// TIA Portal V20 export
// export: Created 2026-07-19T01:14:26.1398018Z, ExportSetting WithDefaults, DisplayName Totally Integrated Automation Portal, DisplayVersion V20 Update 5, DisplayName TIA Portal Openness, DisplayVersion V20 Update 4, DisplayName TIA Portal Version Control Interface, DisplayVersion V20 Update 5, DisplayName SINAMICS Startdrive Advanced, DisplayVersion V20, DisplayName SINAMICS DCC, DisplayVersion V20, DisplayName SINAMICS Startdrive G130, G150, S120, S150, SINAMICS MV, G220, S200, S210, DisplayVersion V20, DisplayName SINAMICS Startdrive G110M, G120, G120C, G120D, G120P, G115D, DisplayVersion V20, DisplayName STEP 7 Professional, DisplayVersion V20 Update 5, DisplayName STEP 7 Safety, DisplayVersion V20 Update 2, DisplayName WinCC Basic/Comfort/Advanced, DisplayVersion V20 Update 5, DisplayName WinCC Unified, DisplayVersion V20 Update 5
FUNCTION "HandAuthorSplitsMerges" : Void   // FC3, LAD
{ S7_Optimized_Access := 'TRUE' }
VERSION : 0.1
// stored: AutoNumber true, IsIECCheckEnabled false, SetENOAutomatically false, UDAEnableTagReadback false
   VAR_OUTPUT
      OutputVars : Array[0..10] of Bool;
   END_VAR
   VAR_TEMP   // added for the SCL form of the ladder/FBD networks
      _w1 : Bool;
      _w2 : Bool;
   END_VAR
BEGIN

REGION Network 1: Split Cascade
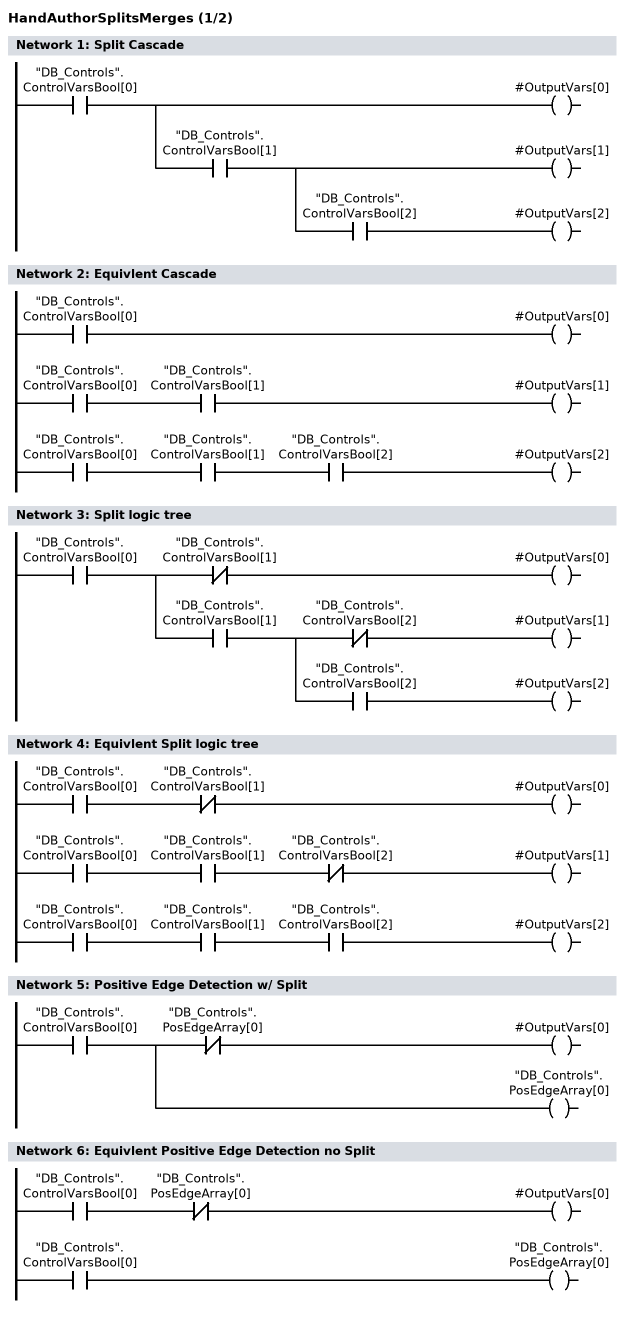
   RUNG wire#powerrail
      Contact( "DB_Controls".ControlVarsBool[0] )
      wire#w1
      Coil( #OutputVars[0] )
   END_RUNG
   RUNG wire#w1
      Contact( "DB_Controls".ControlVarsBool[1] )
      wire#w2
      Coil( #OutputVars[1] )
   END_RUNG
   RUNG wire#w2
      Contact( "DB_Controls".ControlVarsBool[2] )
      Coil( #OutputVars[2] )
   END_RUNG
   // the same network as SCL:
   #OutputVars[0] := "DB_Controls".ControlVarsBool[0];
   #OutputVars[1] := "DB_Controls".ControlVarsBool[0] AND "DB_Controls".ControlVarsBool[1];
   #OutputVars[2] := "DB_Controls".ControlVarsBool[0] AND "DB_Controls".ControlVarsBool[1] AND "DB_Controls".ControlVarsBool[2];
END_REGION

REGION Network 2: Equivlent Cascade
   RUNG wire#powerrail
      Contact( "DB_Controls".ControlVarsBool[0] )
      Coil( #OutputVars[0] )
   END_RUNG
   RUNG wire#powerrail
      Contact( "DB_Controls".ControlVarsBool[0] )
      Contact( "DB_Controls".ControlVarsBool[1] )
      Coil( #OutputVars[1] )
   END_RUNG
   RUNG wire#powerrail
      Contact( "DB_Controls".ControlVarsBool[0] )
      Contact( "DB_Controls".ControlVarsBool[1] )
      Contact( "DB_Controls".ControlVarsBool[2] )
      Coil( #OutputVars[2] )
   END_RUNG
   // the same network as SCL:
   #OutputVars[0] := "DB_Controls".ControlVarsBool[0];
   #OutputVars[1] := "DB_Controls".ControlVarsBool[0] AND "DB_Controls".ControlVarsBool[1];
   #OutputVars[2] := "DB_Controls".ControlVarsBool[0] AND "DB_Controls".ControlVarsBool[1] AND "DB_Controls".ControlVarsBool[2];
END_REGION

REGION Network 3: Split logic tree
   RUNG wire#powerrail
      Contact( "DB_Controls".ControlVarsBool[0] )
      wire#w1
      I_Contact( "DB_Controls".ControlVarsBool[1] )
      Coil( #OutputVars[0] )
   END_RUNG
   RUNG wire#w1
      Contact( "DB_Controls".ControlVarsBool[1] )
      wire#w2
      I_Contact( "DB_Controls".ControlVarsBool[2] )
      Coil( #OutputVars[1] )
   END_RUNG
   RUNG wire#w2
      Contact( "DB_Controls".ControlVarsBool[2] )
      Coil( #OutputVars[2] )
   END_RUNG
   // the same network as SCL:
   #OutputVars[0] := "DB_Controls".ControlVarsBool[0] AND NOT "DB_Controls".ControlVarsBool[1];
   #_w1 := "DB_Controls".ControlVarsBool[0] AND "DB_Controls".ControlVarsBool[1];
   #OutputVars[1] := #_w1 AND NOT "DB_Controls".ControlVarsBool[2];
   #OutputVars[2] := #_w1 AND "DB_Controls".ControlVarsBool[2];
END_REGION

REGION Network 4: Equivlent Split logic tree
   RUNG wire#powerrail
      Contact( "DB_Controls".ControlVarsBool[0] )
      I_Contact( "DB_Controls".ControlVarsBool[1] )
      Coil( #OutputVars[0] )
   END_RUNG
   RUNG wire#powerrail
      Contact( "DB_Controls".ControlVarsBool[0] )
      Contact( "DB_Controls".ControlVarsBool[1] )
      I_Contact( "DB_Controls".ControlVarsBool[2] )
      Coil( #OutputVars[1] )
   END_RUNG
   RUNG wire#powerrail
      Contact( "DB_Controls".ControlVarsBool[0] )
      Contact( "DB_Controls".ControlVarsBool[1] )
      Contact( "DB_Controls".ControlVarsBool[2] )
      Coil( #OutputVars[2] )
   END_RUNG
   // the same network as SCL:
   #OutputVars[0] := "DB_Controls".ControlVarsBool[0] AND NOT "DB_Controls".ControlVarsBool[1];
   #OutputVars[1] := "DB_Controls".ControlVarsBool[0] AND "DB_Controls".ControlVarsBool[1] AND NOT "DB_Controls".ControlVarsBool[2];
   #OutputVars[2] := "DB_Controls".ControlVarsBool[0] AND "DB_Controls".ControlVarsBool[1] AND "DB_Controls".ControlVarsBool[2];
END_REGION

REGION Network 5: Positive Edge Detection w/ Split
   RUNG wire#powerrail
      Contact( "DB_Controls".ControlVarsBool[0] )
      wire#w1
      I_Contact( "DB_Controls".PosEdgeArray[0] )
      Coil( #OutputVars[0] )
   END_RUNG
   RUNG wire#w1
      Coil( "DB_Controls".PosEdgeArray[0] )
   END_RUNG
   // the same network as SCL:
   #OutputVars[0] := "DB_Controls".ControlVarsBool[0] AND NOT "DB_Controls".PosEdgeArray[0];
   "DB_Controls".PosEdgeArray[0] := "DB_Controls".ControlVarsBool[0];
END_REGION

REGION Network 6: Equivlent Positive Edge Detection no Split
   RUNG wire#powerrail
      Contact( "DB_Controls".ControlVarsBool[0] )
      I_Contact( "DB_Controls".PosEdgeArray[0] )
      Coil( #OutputVars[0] )
   END_RUNG
   RUNG wire#powerrail
      Contact( "DB_Controls".ControlVarsBool[0] )
      Coil( "DB_Controls".PosEdgeArray[0] )
   END_RUNG
   // the same network as SCL:
   #OutputVars[0] := "DB_Controls".ControlVarsBool[0] AND NOT "DB_Controls".PosEdgeArray[0];
   "DB_Controls".PosEdgeArray[0] := "DB_Controls".ControlVarsBool[0];
END_REGION

REGION Network 7: Negitive Edge Detection /w split and merge
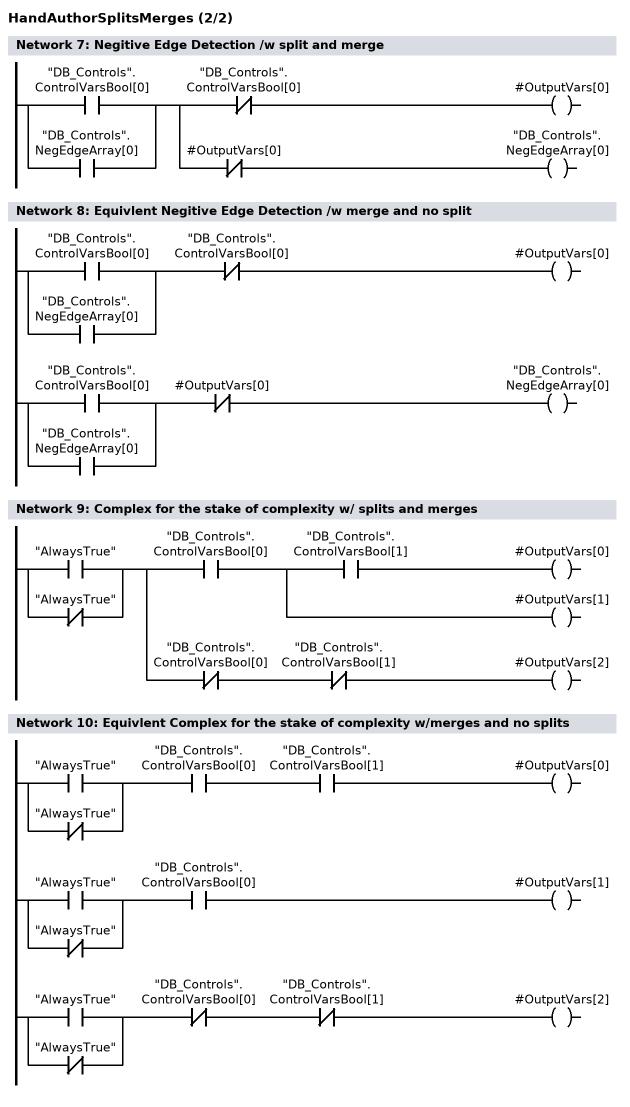
   RUNG wire#powerrail
      Contact( "DB_Controls".ControlVarsBool[0] )
      wire#w1
      I_Contact( "DB_Controls".ControlVarsBool[0] )
      Coil( #OutputVars[0] )
   END_RUNG
   RUNG wire#powerrail
      Contact( "DB_Controls".NegEdgeArray[0] )
   END_RUNG wire#w1
   RUNG wire#w1
      I_Contact( #OutputVars[0] )
      Coil( "DB_Controls".NegEdgeArray[0] )
   END_RUNG
   // the same network as SCL:
   #_w1 := "DB_Controls".ControlVarsBool[0] OR "DB_Controls".NegEdgeArray[0];
   #OutputVars[0] := #_w1 AND NOT "DB_Controls".ControlVarsBool[0];
   "DB_Controls".NegEdgeArray[0] := #_w1 AND NOT #OutputVars[0];
END_REGION

REGION Network 8: Equivlent Negitive Edge Detection /w merge and no split
   RUNG wire#powerrail
      Contact( "DB_Controls".ControlVarsBool[0] )
      wire#w1
      I_Contact( "DB_Controls".ControlVarsBool[0] )
      Coil( #OutputVars[0] )
   END_RUNG
   RUNG wire#powerrail
      Contact( "DB_Controls".NegEdgeArray[0] )
   END_RUNG wire#w1
   RUNG wire#powerrail
      Contact( "DB_Controls".ControlVarsBool[0] )
      wire#w2
      I_Contact( #OutputVars[0] )
      Coil( "DB_Controls".NegEdgeArray[0] )
   END_RUNG
   RUNG wire#powerrail
      Contact( "DB_Controls".NegEdgeArray[0] )
   END_RUNG wire#w2
   // the same network as SCL:
   #OutputVars[0] := ("DB_Controls".ControlVarsBool[0] OR "DB_Controls".NegEdgeArray[0]) AND NOT "DB_Controls".ControlVarsBool[0];
   "DB_Controls".NegEdgeArray[0] := ("DB_Controls".ControlVarsBool[0] OR "DB_Controls".NegEdgeArray[0]) AND NOT #OutputVars[0];
END_REGION

REGION Network 9: Complex for the stake of complexity w/ splits and merges
   RUNG wire#powerrail
      Contact( "AlwaysTrue" )
      wire#w1
      Contact( "DB_Controls".ControlVarsBool[0] )
      wire#w2
      Contact( "DB_Controls".ControlVarsBool[1] )
      Coil( #OutputVars[0] )
   END_RUNG
   RUNG wire#powerrail
      I_Contact( "AlwaysTrue" )
   END_RUNG wire#w1
   RUNG wire#w2
      Coil( #OutputVars[1] )
   END_RUNG
   RUNG wire#w1
      I_Contact( "DB_Controls".ControlVarsBool[0] )
      I_Contact( "DB_Controls".ControlVarsBool[1] )
      Coil( #OutputVars[2] )
   END_RUNG
   // the same network as SCL:
   #_w1 := "AlwaysTrue" OR NOT "AlwaysTrue";
   #_w2 := #_w1 AND "DB_Controls".ControlVarsBool[0];
   #OutputVars[0] := #_w2 AND "DB_Controls".ControlVarsBool[1];
   #OutputVars[1] := #_w2;
   #OutputVars[2] := #_w1 AND NOT "DB_Controls".ControlVarsBool[0] AND NOT "DB_Controls".ControlVarsBool[1];
END_REGION

REGION Network 10: Equivlent Complex for the stake of complexity w/merges and no splits
   RUNG wire#powerrail
      Contact( "AlwaysTrue" )
      wire#w1
      Contact( "DB_Controls".ControlVarsBool[0] )
      Contact( "DB_Controls".ControlVarsBool[1] )
      Coil( #OutputVars[0] )
   END_RUNG
   RUNG wire#powerrail
      I_Contact( "AlwaysTrue" )
   END_RUNG wire#w1
   RUNG wire#powerrail
      Contact( "AlwaysTrue" )
      wire#w2
      Contact( "DB_Controls".ControlVarsBool[0] )
      Coil( #OutputVars[1] )
   END_RUNG
   RUNG wire#powerrail
      I_Contact( "AlwaysTrue" )
   END_RUNG wire#w2
   RUNG wire#powerrail
      Contact( "AlwaysTrue" )
      wire#w3
      I_Contact( "DB_Controls".ControlVarsBool[0] )
      I_Contact( "DB_Controls".ControlVarsBool[1] )
      Coil( #OutputVars[2] )
   END_RUNG
   RUNG wire#powerrail
      I_Contact( "AlwaysTrue" )
   END_RUNG wire#w3
   // the same network as SCL:
   #OutputVars[0] := ("AlwaysTrue" OR NOT "AlwaysTrue") AND "DB_Controls".ControlVarsBool[0] AND "DB_Controls".ControlVarsBool[1];
   #OutputVars[1] := ("AlwaysTrue" OR NOT "AlwaysTrue") AND "DB_Controls".ControlVarsBool[0];
   #OutputVars[2] := ("AlwaysTrue" OR NOT "AlwaysTrue") AND NOT "DB_Controls".ControlVarsBool[0] AND NOT "DB_Controls".ControlVarsBool[1];
END_REGION
END_FUNCTION
